PROGRAM Rotation_Sample
VAR
END_VAR

astAxes[AXIS_ROTATION_SAMPLE].stControl.bEnable := TRUE;
astAxes[AXIS_ROTATION_SAMPLE].stInputs.bLimitBwd := astAxes[AXIS_ROTATION].stInputs.bLimitBwd;
astAxes[AXIS_ROTATION_SAMPLE].stInputs.bLimitFwd := astAxes[AXIS_ROTATION].stInputs.bLimitFwd;

astAxes[AXIS_ROTATION_SAMPLE].stDescription.sAxisName := 'SAMPLE_ROT';

END_PROGRAM

(* stored: Version 1.1.0.1, ProductVersion 3.1.4024.12
   POU Rotation_Sample: Id {db16538d-0000-497f-bb9f-c95fd0b6faff}, SpecialFunc None *)
